# EPICS substitutions: CONEXAGP/CONEXAGP-IOC-01App/Db/asyn_motor.substitutions
file $(MOTOR)/motorApp/Db/asyn_motor.db {

pattern {P,    N,   M,         DTYP,        PORT, ADDR,         DESC,   EGU,  DIR,  VELO,  VBAS, ACCL, BDST, BVEL, BACC,    MRES, PREC, DHLM, DLLM, INIT}
{"\$(P)", 1, "\$(M)", "asynMotor",  "\$(PORT)",    "\$(ADDR)", "Horizontal",    mm,  Pos,    .5,   0.1,  .25,    0,    1,   .2,   .0001,    4,   28,   -1,   ""}

}
